PROGRAM MAIN
VAR
	
	//Pulsador AT %I*: BOOL;
	//Lampara AT %Q*: BOOL;
	
	Estacion: FB_Estacion;

END_VAR

Estacion();

END_PROGRAM

(* stored: Version 1.1.0.1, ProductVersion 3.1.4024.12
   POU MAIN: Id {00882189-f86f-4cea-921e-f5fd8e9f7b86}, SpecialFunc None *)
